// TwinCAT 3 PLC project Pers
// ProgramVersion: 3.1.4022.3
// libraries:
//   Tc2_Standard, * (Beckhoff Automation GmbH)
//   Tc2_System, * (Beckhoff Automation GmbH)
//   Tc3_Module, * (Beckhoff Automation GmbH)
// project tree:
//   DUTs/ Pers_Struct.TcDUT
//   GVLs/ GVL_Pers.TcGVL, GVL_Non_Pers.TcGVL
//   / PlcTask.TcTTO
//   POUs/ MAIN.TcPOU
// real-time tasks:
//   TASK PlcTask: cycle T#10ms, priority 20, ADS port 350

CONFIGURATION Pers
    RESOURCE PLC ON TwinCAT3
        TASK PlcTask(INTERVAL := T#10ms, PRIORITY := 20);
        PROGRAM MAIN WITH PlcTask : MAIN;
    END_RESOURCE
END_CONFIGURATION

// ---- DUTs/Pers_Struct.TcDUT
TYPE Pers_Struct :
STRUCT
	int1 : INT;
	bool1 : BOOL;
END_STRUCT
END_TYPE

// ---- GVLs/GVL_Pers.TcGVL
{attribute 'qualified_only'}
VAR_GLOBAL PERSISTENT
	testPeristent: INT;
	test_Struct_Pers : Pers_Struct;
END_VAR

// ---- GVLs/GVL_Non_Pers.TcGVL
{attribute 'qualified_only'}
VAR_GLOBAL
	testNonPers : INT;
END_VAR

// ---- POUs/MAIN.TcPOU
PROGRAM MAIN
VAR
END_VAR

GVL_Pers.testPeristent := GVL_Pers.testPeristent +10;
GVL_Non_Pers.testNonPers := GVL_Non_Pers.testNonPers +10;

END_PROGRAM
